// TIA Portal V20 export
DATA_BLOCK "IDB_EmptyLine"   // DB9
// stored: InstanceOfName EmptyLine.FB_EmptyLine, InstanceOfType FB, Namespace EmptyLine
"EmptyLine.FB_EmptyLine"
   // VAR
   //    "J1.1.1" : "Global.FB_Conveyor";
   //    "J1.1.2" { S7_SetPoint := 'True'} : "Global.FB_Conveyor";
   //    "J1.1.3" { S7_SetPoint := 'True'} : "Global.FB_Conveyor";
   //    "J1.1.4" { S7_SetPoint := 'True'} : "Global.FB_Conveyor";
   //    "J1.1.5" { S7_SetPoint := 'True'} : "Global.FB_Conveyor";
   //    "J1.1.6" { S7_SetPoint := 'True'} : "Global.FB_Conveyor";
   //    "J1.1.7" { S7_SetPoint := 'True'} : "Global.FB_Conveyor";
   //    "J1.1.8" { S7_SetPoint := 'True'} : "Global.FB_Conveyor";
   //    "J1.1.9" { S7_SetPoint := 'True'} : "Global.FB_Conveyor";
   //    "J1.1.10" { S7_SetPoint := 'True'} : "Global.FB_Conveyor";
   //    "J1.1.11" { S7_SetPoint := 'True'} : "Global.FB_Conveyor";
   //    "J1.1.12" { S7_SetPoint := 'True'} : "Global.FB_Conveyor";
   //    "J1.1.13" { S7_SetPoint := 'True'} : "Global.FB_Conveyor";
   //    "J1.1.14" { S7_SetPoint := 'True'} : "Global.FB_Conveyor";
   //    "J1.1.15" { S7_SetPoint := 'True'} : "Global.FB_Conveyor";
   //    "J1.1.16" { S7_SetPoint := 'True'} : "Global.FB_Conveyor";
   //    "J1.2.1" { S7_SetPoint := 'True'} : "Global.FB_Conveyor";
   //    "J1.2.2" { S7_SetPoint := 'True'} : "Global.FB_Conveyor";
   //    "J1.2.3" { S7_SetPoint := 'True'} : "Global.FB_Conveyor";
   //    "J2.1.1" { S7_SetPoint := 'True'} : "Global.FB_Conveyor";
   //    "J2.1.2" { S7_SetPoint := 'True'} : "Global.FB_Conveyor";
   //    "J2.1.3" { S7_SetPoint := 'True'} : "Global.FB_Conveyor";
   //    "J2.1.4" { S7_SetPoint := 'True'} : "Global.FB_Conveyor";
   //    "J2.1.5" { S7_SetPoint := 'True'} : "Global.FB_Conveyor";
   //    "J2.1.6" { S7_SetPoint := 'True'} : "Global.FB_Conveyor";
   //    "J2.1.7" { S7_SetPoint := 'True'} : "Global.FB_Conveyor";
   //    "J2.1.8" { S7_SetPoint := 'True'} : "Global.FB_Conveyor";
   //    "J2.1.9" { S7_SetPoint := 'True'} : "Global.FB_Conveyor";
   //    "J2.1.10" { S7_SetPoint := 'True'} : "Global.FB_Conveyor";
   //    "J2.1.11" { S7_SetPoint := 'True'} : "Global.FB_Conveyor";
   //    "J2.1.12" { S7_SetPoint := 'True'} : "Global.FB_Conveyor";
   //    "J2.1.13" { S7_SetPoint := 'True'} : "Global.FB_Conveyor";
   //    "J2.1.14" { S7_SetPoint := 'True'} : "Global.FB_Conveyor";
   //    "J2.1.15" { S7_SetPoint := 'True'} : "Global.FB_Conveyor";
   //    "J2.2.1" { S7_SetPoint := 'True'} : "Global.FB_Conveyor";
   //    "J2.2.2" { S7_SetPoint := 'True'} : "Global.FB_Conveyor";
   //    "J2.3.1" { S7_SetPoint := 'True'} : "Global.FB_Conveyor";
   //    "J2.4.1" { S7_SetPoint := 'True'} : "Global.FB_Conveyor";
   //    "J1.2.4" { S7_SetPoint := 'True'} : "Global.FB_Conveyor";
   //    "J1.2.5" { S7_SetPoint := 'True'} : "Global.FB_Conveyor";
   //    "J1.3.1" { S7_SetPoint := 'True'} : "Global.FB_Conveyor";
   //    "J1.3.2" { S7_SetPoint := 'True'} : "Global.FB_Conveyor";
   //    "J1.4.1" { S7_SetPoint := 'True'} : "Global.FB_Conveyor";
   //    "J1.4.2" { S7_SetPoint := 'True'} : "Global.FB_Conveyor";
   //    "J1.4.3" { S7_SetPoint := 'True'} : "Global.FB_Conveyor";
   //    "J1.4.4" { S7_SetPoint := 'True'} : "Global.FB_Conveyor";
   //    "J1.4.5" { S7_SetPoint := 'True'} : "Global.FB_Conveyor";
   //    "J1.4.6" { S7_SetPoint := 'True'} : "Global.FB_Conveyor";
   //    "J1.4.7" { S7_SetPoint := 'True'} : "Global.FB_Conveyor";
   //    "J1.5.1" { S7_SetPoint := 'True'} : "Global.FB_Conveyor";
   //    "J1.5.2" { S7_SetPoint := 'True'} : "Global.FB_Conveyor";
   //    "J1.5.3" { S7_SetPoint := 'True'} : "Global.FB_Conveyor";
   //    "J1.5.4" { S7_SetPoint := 'True'} : "Global.FB_Conveyor";
   //    "J1.6.1" { S7_SetPoint := 'True'} : "Global.FB_MABS";
   //    "J1.6.2" { S7_SetPoint := 'True'} : "Global.FB_MABS";
   //    "J1.7.1" { S7_SetPoint := 'True'} : "Global.FB_Conveyor";
   //    "J1.7.2" { S7_SetPoint := 'True'} : "Global.FB_Conveyor";
   //    "J1.8.1" { S7_SetPoint := 'True'} : "Global.FB_Conveyor";
   //    "J1.8.2" { S7_SetPoint := 'True'} : "Global.FB_Conveyor";
   //    "J1.9.1" { S7_SetPoint := 'True'} : "Global.FB_Conveyor";
   //    "J1.10.1" { S7_SetPoint := 'True'} : "Global.FB_Conveyor";
   //    "J1.11.1" { S7_SetPoint := 'True'} : "Global.FB_Conveyor";
   //    "J1.11.2" { S7_SetPoint := 'True'} : "Global.FB_Conveyor";
   //    "J1.11.3" { S7_SetPoint := 'True'} : "Global.FB_Conveyor";
   //    "J1.11.4" { S7_SetPoint := 'True'} : "Global.FB_Conveyor";
   //    "J1.11.5" { S7_SetPoint := 'True'} : "Global.FB_Conveyor";
   //    "J1.11.6" { S7_SetPoint := 'True'} : "Global.FB_Conveyor";
   //    "J1.11.7" { S7_SetPoint := 'True'} : "Global.FB_Conveyor";
   //    "J1.11.8" { S7_SetPoint := 'True'} : "Global.FB_Conveyor";
   //    "J1.11.9" { S7_SetPoint := 'True'} : "Global.FB_Conveyor";
   //    "J1.11.10" { S7_SetPoint := 'True'} : "Global.FB_Conveyor";
   //    "J1.11.11" { S7_SetPoint := 'True'} : "Global.FB_Conveyor";
   //    "J1.11.12" { S7_SetPoint := 'True'} : "Global.FB_Conveyor";
   //    "J1.11.13" { S7_SetPoint := 'True'} : "Global.FB_Conveyor";
   //    "K1.1.1" { S7_SetPoint := 'True'} : "Global.FB_Conveyor";
   //    "K1.2.1" { S7_SetPoint := 'True'} : "Global.FB_Conveyor";
   //    "K1.3.1" { S7_SetPoint := 'True'} : "Global.FB_Conveyor";
   //    "K1.4.1" { S7_SetPoint := 'True'} : "Global.FB_Conveyor";
   //    "K1.4.2" { S7_SetPoint := 'True'} : "Global.FB_Conveyor";
   //    "K1.4.3" { S7_SetPoint := 'True'} : "Global.FB_Conveyor";
   //    "K1.4.4" { S7_SetPoint := 'True'} : "Global.FB_Conveyor";
   //    "K1.4.5" { S7_SetPoint := 'True'} : "Global.FB_Conveyor";
   //    "K1.4.6" { S7_SetPoint := 'True'} : "Global.FB_Conveyor";
   //    "K1.4.7" { S7_SetPoint := 'True'} : "Global.FB_Conveyor";
   //    "K1.4.8" { S7_SetPoint := 'True'} : "Global.FB_Conveyor";
   //    "K1.4.9" { S7_SetPoint := 'True'} : "Global.FB_Conveyor";
   //    "K1.4.10" { S7_SetPoint := 'True'} : "Global.FB_Conveyor";
   //    "K1.5.1" { S7_SetPoint := 'True'} : "Global.FB_Conveyor";
   //    "K1.5.2" { S7_SetPoint := 'True'} : "Global.FB_Conveyor";
   //    "K1.5.3" { S7_SetPoint := 'True'} : "Global.FB_Conveyor";
   //    "K1.5.4" { S7_SetPoint := 'True'} : "Global.FB_Conveyor";
   //    "K1.5.5" { S7_SetPoint := 'True'} : "Global.FB_Conveyor";
   //    "K1.5.6" { S7_SetPoint := 'True'} : "Global.FB_Conveyor";
   //    "K1.5.7" { S7_SetPoint := 'True'} : "Global.FB_Conveyor";
   //    "K1.5.8" { S7_SetPoint := 'True'} : "Global.FB_Conveyor";
   //    "K1.6.1" { S7_SetPoint := 'True'} : "Global.FB_Conveyor";
   //    "K1.6.2" { S7_SetPoint := 'True'} : "Global.FB_Conveyor";
   //    "K1.7.1" { S7_SetPoint := 'True'} : "Global.FB_Conveyor";
   //    "K1.7.2" { S7_SetPoint := 'True'} : "Global.FB_Conveyor";
   //    "K1.8.1" { S7_SetPoint := 'True'} : "Global.FB_Conveyor";
   //    "K1.8.2" { S7_SetPoint := 'True'} : "Global.FB_Conveyor";
   //    "K1.8.3" { S7_SetPoint := 'True'} : "Global.FB_Conveyor";
   //    "K1.9.1" { S7_SetPoint := 'True'} : "Global.FB_Conveyor";
   //    "K1.9.2" { S7_SetPoint := 'True'} : "Global.FB_Conveyor";
   //    "K1.9.3" { S7_SetPoint := 'True'} : "Global.FB_Conveyor";
   //    "K1.9.4" { S7_SetPoint := 'True'} : "Global.FB_Conveyor";
   //    "K1.9.5" { S7_SetPoint := 'True'} : "Global.FB_Conveyor";
   //    "K1.9.6" { S7_SetPoint := 'True'} : "Global.FB_Conveyor";
   //    "K1.9.7" { S7_SetPoint := 'True'} : "Global.FB_Conveyor";
   //    "K1.10.1" { S7_SetPoint := 'True'} : "Global.FB_Conveyor";
   // END_VAR
BEGIN
END_DATA_BLOCK
